{attribute 'Tc2GvlVarNames'}
VAR_GLOBAL

(*TERMINAL XXXKF1 - EK1100 **********************************************************)

(*TERMINAL 350KF1 (EL6001 Interface (RS232))  ********1-Channel Serial Interface RS232***********************)
	ib350A1_EL6001PortNo								AT %I* :  UINT;
	ist350A1_HandScannerCOMPortDataIn					AT %I* :  EL6InData22B;
	qst350A1_HandScannerCOMPortDataOut					AT %Q*: EL6OutData22B;

(*TERMINAL 351KF1 - EL4002 ******************************************************)
	qn351KF1_1_OuterValidationLightingIntensity			AT %Q* : INT;
	qn351KF1_2_OuterAggregationLightingIntensity		AT %Q* : INT;

(*TERMINAL 352KF1 - EL4002 ******************************************************)
	qn352KF1_1_CaseContentValidationLightingIntensity	AT %Q* : INT;
	qn352KF1_2_LightingIntensity							AT %Q* : INT;

(*TERMINAL 360KF1 - EL1008 ***********************************************************)
	ib360KF1_1_OuterAtInfeed							AT %I* : BOOL;	(* Option *)
	ib360KF1_5_OuterInfeedBlocked						AT %I* : BOOL;	(* Option clamp*)
	ib360KF1_2_OuterAtLabeller							AT %I* : BOOL;	(* Option gate*)
	ib360KF1_6_PackConfirmationCameraTrigSensor			AT %I* : BOOL;
	ib360KF1_3_OuterValidationCameraTrigSensor 					AT %I* : BOOL;
	ib360KF1_7_OuterAtReject							AT %I* : BOOL;
	ib360KF1_4_RejectConfirmation						AT %I* : BOOL;
	ib360KF1_8_RejectBinFull								AT %I* : BOOL;

(*TERMINAL 361KF1 - EL1008 ***********************************************************)
	ib361KF1_1_OuterClampExtended							AT %I* : BOOL;
	ib361KF1_5_OuterGateExtended					AT %I* : BOOL;
	ib361KF1_2_OuterGateRetracted						AT %I* : BOOL;
	ib361KF1_6_OuterGateImpactSensor						AT %I* : BOOL;
	ib361KF1_3_RejectCylinderExtended					AT %I* : BOOL;
	ib361KF1_7_RejectCylinderRetracted					AT %I* : BOOL;
	ib361KF1_4_EUCAExitBlocked										AT %I* : BOOL;	(* Option *)
	ib361KF1_8_EUCABuildBack									AT %I* : BOOL;

(*TERMINAL 362KF1 - EL1008 ************************************************************)
	ib362KF1_1_Labeller02Ready							AT %I*: BOOL;
	ib362KF1_5_Labeller02DataReady						AT %I*: BOOL;
	ib362KF1_2_Labeller02HomePosition 			AT %I*: BOOL;
	ib362KF1_6_Labeller02LabelPrinted						AT %I*: BOOL;
	ib362KF1_3_Labeller02SummaryWarning					AT %I*: BOOL;
	ib362KF1_7_Labeller02Error							AT %I*: BOOL;
	ib362KF1_4_Labeller02AirPressureOK							AT %I*: BOOL;
	ib362KF1_8_Labeller02InPosition					AT %I*: BOOL;	(* ??? *)

(*TERMINAL 363KF1 (EL1008 8Ch. Dig. Input 24V, 3ms) ***************************************)
	ib363KF1_1_QAButtonRejectOuter						AT %I*: BOOL;	(* Option *)
	ib363KF1_5_IntermediatePushSensor					AT %I*: BOOL;
	ib363KF1_2_CaseLabelValidationCameraTrigSensor 		AT %I*: BOOL;
	ib363KF1_6_OuterAggregationCameraTrigSensor			AT %I*: BOOL;	(* *)
	ib363KF1_3_RowCompleteSensor						AT %I*: BOOL;
	ib363KF1_7_LayerCompleteSensor						AT %I*: BOOL;
	ib363KF1_4_CaseCompleteSensor						AT %I*: BOOL;
	ib363KF1_8_CaseDischargedSensor						AT %I*: BOOL;

(*TERMINAL 366KF1 (EL1008 8Ch. Dig. Input 24V, 3ms) ****************************************)
	ib366KF1_1_OuterAtAdditionalConveyor02									AT %I*: BOOL;
	ib366KF1_5_ExitBlockedAdditionalConveyor02									AT %I*: BOOL;
	ib366KF1_2_Spare									AT %I*: BOOL;
	ib366KF1_6_Spare									AT %I*: BOOL;
	ib366KF1_3_Spare									AT %I*: BOOL;
	ib366KF1_7_Spare									AT %I*: BOOL;
	ib366KF1_4_Spare								AT %I*: BOOL;
	ib366KF1_8_RemoteAirSupplyOK									AT %I*: BOOL;

(*TERMINAL 380KF1 - EL2008 (EL2008 8Ch. Dig. Output 24V, 0.5A) ********************************)
	qb380KF1_1_ClampCylinderExtend				AT %Q*: BOOL;
	qb380KF1_5_Spare						 			AT %Q*: BOOL;
	qb380KF1_2_GateCylinderExtend 						AT %Q*: BOOL;		(**)
	qb380KF1_6_GateCylinderRetract	 					AT %Q*: BOOL;		(**)
	qb380KF1_3_RejectCylinderExtend						AT %Q*: BOOL;
	qb380KF1_7_RejectCylinderRetract			  		AT %Q*: BOOL;
	qb380KF1_4_Spare								AT %Q*: BOOL;
	qb380KF1_8_PLCControlledAggCameraLightning			AT %Q*: BOOL; (**)

(*TERMINAL 381KF1 (EL2008 8Ch. Dig. Output 24V, 0.5A) ***************************************)
	qb381KF1_1_RearConfirmationCameraTrigger			AT %Q*: BOOL;
	qb381KF1_5_RearConfirmationCameraPower				AT %Q*: BOOL;
	qb381KF1_2_FrontConfirmationCameraTrigger			AT %Q*: BOOL;
	qb381KF1_6_FrontConfirmationCameraPower	 			AT %Q*: BOOL;
	qb381KF1_3_OuterValidationCameraTrig 					AT %Q*: BOOL;
	qb381KF1_7_OuterValidationCameraPower				AT %Q*: BOOL;
	qb381KF1_4_OuterAggregationCameraTrig					AT %Q*: BOOL;
	qb381KF1_8_OuterAggregationCameraPower					AT %Q*: BOOL;

(*TERMINAL 382KF1 (EL2008 8Ch. Dig. Output 24V, 0.5A) ****************************************)
	qb382KF1_1_CaseContentValidationCameraTrig				AT %Q*: BOOL;
	qb382KF1_5_CaseContentValidationCameraPower			AT %Q*: BOOL;
	qb382KF1_2_CaseLabelValidationCameraTrig				AT %Q*: BOOL;
	qb382KF1_6_CaseLabelValidationCameraPower	 			AT %Q*: BOOL;
	qb382KF1_3_OuterValidationCameraLightning					AT %Q*: BOOL;		(**)
	qb382KF1_7_OuterAggregationCameraLightning				AT %Q*: BOOL;		(**)
	qb382KF1_4_CaseContentValidationCameraLightning			AT %Q*: BOOL;		(**)
	qb382KF1_8_Labeller02DoorGuardOpen				AT %Q*: BOOL;		(**)

(*TERMINAL 390KF1 (EL2624 4Ch. Relay Output, 125 V AC, 30 V DC, 0.5 A AC, 2 A DC)******************)
	qb390KF1_1_Labeller02ResetSignal						AT %Q*: BOOL;
	qb390KF1_2_Labeller02PrintSignal						AT %Q*: BOOL;
	qb390KF1_3_Labeller02ApplySignal1						AT %Q*: BOOL;
	qb390KF1_4_Labeller02ApplySignal2								AT %Q*: BOOL;

END_VAR

(* stored: Version 1.1.0.1, ProductVersion 3.1.4024.15
   GVL IOVariablesEUCA_OC: Id {a76442b3-e20b-4ac1-9801-fcb0123a43f0} *)
